INTERFACE I_Switchable

PROPERTY Active : BOOL
GET
END_GET
END_PROPERTY

METHOD Off : BOOL
VAR_INPUT
END_VAR
END_METHOD

METHOD On : BOOL
VAR_INPUT
END_VAR
END_METHOD

END_INTERFACE

(* stored: Version 1.1.0.1, ProductVersion 3.1.4024.5
   Itf I_Switchable: Id {29d91e68-88a3-4fc7-bfbf-5e03920843bf}
   Property Active: Id {6f11b715-3331-4f72-bc39-07e3410fcdd5}
   Get Get: Id {fc206d9b-003c-41a9-aa8e-2cb979bff0e1}
   Method Off: Id {e385c2c4-956e-4ee3-98ad-8907da012b89}
   Method On: Id {84093c63-3f32-49a5-896b-aaa987fea412} *)
